Staubli VAL3: setVelocity.pgx

public program setVelocity(num x_nValue, num x_nIndex)
begin
  nVelocity[x_nIndex]=x_nValue
end
